// TIA Portal V17 program export: 2 tag tables, 2 data types, 1 data blocks, 3 code blocks (in call order from the OBs), 2 instance data blocks

VAR_GLOBAL   // PLC tag table "Default tag table"
   Clock_Byte AT %MB0 : Byte;
   Clock_10Hz AT %M0.0 : Bool;
   Clock_5Hz AT %M0.1 : Bool;
   "Clock_2.5Hz" AT %M0.2 : Bool;
   Clock_2Hz AT %M0.3 : Bool;
   "Clock_1.25Hz" AT %M0.4 : Bool;
   Clock_1Hz AT %M0.5 : Bool;
   "Clock_0.625Hz" AT %M0.6 : Bool;
   "Clock_0.5Hz" AT %M0.7 : Bool;
END_VAR

VAR_GLOBAL   // PLC tag table "OPC_StatusCodes"
END_VAR
VAR_GLOBAL CONSTANT   // user constants
   OpcUa_Good : DWord := 16#00000000;   // Everything is as expected.
   OpcUa_Uncertain : DWord := 16#40000000;   // Something unexpected occurred but the results still maybe useable.
   OpcUa_Bad : DWord := 16#80000000;   // An error occurred.
   OpcUa_BadUnexpectedError : DWord := 16#80010000;   // An unexpected error occurred.
   OpcUa_BadInternalError : DWord := 16#80020000;   // An internal error occurred as a result of a programming or configuration error.
   OpcUa_BadOutOfMemory : DWord := 16#80030000;   // Not enough memory to complete the operation.
   OpcUa_BadResourceUnavailable : DWord := 16#80040000;   // An operating system resource is not available.
   OpcUa_BadCommunicationError : DWord := 16#80050000;   // A low level communication error occurred.
   OpcUa_BadEncodingError : DWord := 16#80060000;   // Encoding halted because of invalid data in the objects being serialized.
   OpcUa_BadDecodingError : DWord := 16#80070000;   // Decoding halted because of invalid data in the stream.
   OpcUa_BadEncodingLimitsExceeded : DWord := 16#80080000;   // The message encoding/decoding limits imposed by the stack have been exceeded.
   OpcUa_BadRequestTooLarge : DWord := 16#80B80000;   // The request message size exceeds limits set by the server.
   OpcUa_BadResponseTooLarge : DWord := 16#80B90000;   // The response message size exceeds limits set by the client.
   OpcUa_BadUnknownResponse : DWord := 16#80090000;   // An unrecognized response was received from the server.
   OpcUa_BadTimeout : DWord := 16#800A0000;   // The operation timed out.
   OpcUa_BadServiceUnsupported : DWord := 16#800B0000;   // The server does not support the requested service.
   OpcUa_BadShutdown : DWord := 16#800C0000;   // The operation was cancelled because the application is shutting down.
   OpcUa_BadServerNotConnected : DWord := 16#800D0000;   // The operation could not complete because the client is not connected to the server.
   OpcUa_BadServerHalted : DWord := 16#800E0000;   // The server has stopped and cannot process any requests.
   OpcUa_BadNothingToDo : DWord := 16#800F0000;   // There was nothing to do because the client passed a list of operations with no elements.
   OpcUa_BadTooManyOperations : DWord := 16#80100000;   // The request could not be processed because it specified too many operations.
   OpcUa_BadTooManyMonitoredItems : DWord := 16#80DB0000;   // The request could not be processed because there are too many monitored items in the subscription.
   OpcUa_BadDataTypeIdUnknown : DWord := 16#80110000;   // The extension object cannot be (de)serialized because the data type id is not recognized.
   OpcUa_BadCertificateInvalid : DWord := 16#80120000;   // The certificate provided as a parameter is not valid.
   OpcUa_BadSecurityChecksFailed : DWord := 16#80130000;   // An error occurred verifying security.
   OpcUa_BadCertificateTimeInvalid : DWord := 16#80140000;   // The certificate has expired or is not yet valid.
   OpcUa_BadCertificateIssuerTimeInvalid : DWord := 16#80150000;   // An issuer certificate has expired or is not yet valid.
   OpcUa_BadCertificateHostNameInvalid : DWord := 16#80160000;   // The HostName used to connect to a server does not match a HostName in the certificate.
   OpcUa_BadCertificateUriInvalid : DWord := 16#80170000;   // The URI specified in the ApplicationDescription does not match the URI in the certificate.
   OpcUa_BadCertificateUseNotAllowed : DWord := 16#80180000;   // The certificate may not be used for the requested operation.
   OpcUa_BadCertificateIssuerUseNotAllowed : DWord := 16#80190000;   // The issuer certificate may not be used for the requested operation.
   OpcUa_BadCertificateUntrusted : DWord := 16#801A0000;   // The certificate is not trusted.
   OpcUa_BadCertificateRevocationUnknown : DWord := 16#801B0000;   // It was not possible to determine if the certificate has been revoked.
   OpcUa_BadCertificateIssuerRevocationUnknown : DWord := 16#801C0000;   // It was not possible to determine if the issuer certificate has been revoked.
   OpcUa_BadCertificateRevoked : DWord := 16#801D0000;   // The certificate has been revoked.
   OpcUa_BadCertificateIssuerRevoked : DWord := 16#801E0000;   // The issuer certificate has been revoked.
   OpcUa_BadCertificateChainIncomplete : DWord := 16#810D0000;   // The certificate chain is incomplete.
   OpcUa_BadUserAccessDenied : DWord := 16#801F0000;   // User does not have permission to perform the requested operation.
   OpcUa_BadIdentityTokenInvalid : DWord := 16#80200000;   // The user identity token is not valid.
   OpcUa_BadIdentityTokenRejected : DWord := 16#80210000;   // The user identity token is valid but the server has rejected it.
   OpcUa_BadSecureChannelIdInvalid : DWord := 16#80220000;   // The specified secure channel is no longer valid.
   OpcUa_BadInvalidTimestamp : DWord := 16#80230000;   // The timestamp is outside the range allowed by the server.
   OpcUa_BadNonceInvalid : DWord := 16#80240000;   // The nonce does appear to be not a random value or it is not the correct length.
   OpcUa_BadSessionIdInvalid : DWord := 16#80250000;   // The session id is not valid.
   OpcUa_BadSessionClosed : DWord := 16#80260000;   // The session was closed by the client.
   OpcUa_BadSessionNotActivated : DWord := 16#80270000;   // The session cannot be used because ActivateSession has not been called.
   OpcUa_BadSubscriptionIdInvalid : DWord := 16#80280000;   // The subscription id is not valid.
   OpcUa_BadRequestHeaderInvalid : DWord := 16#802A0000;   // The header for the request is missing or invalid.
   OpcUa_BadTimestampsToReturnInvalid : DWord := 16#802B0000;   // The timestamps to return parameter is invalid.
   OpcUa_BadRequestCancelledByClient : DWord := 16#802C0000;   // The request was cancelled by the client.
   OpcUa_BadTooManyArguments : DWord := 16#80E50000;   // Too many arguments were provided.
   OpcUa_BadLicenseExpired : DWord := 16#810E0000;   // The server requires a license to operate in general or to perform a service or operation, but existing license is expired.
   OpcUa_BadLicenseLimitsExceeded : DWord := 16#810F0000;   // The server has limits on number of allowed operations / objects, based on installed licenses, and these limits where exceeded.
   OpcUa_BadLicenseNotAvailable : DWord := 16#81100000;   // The server does not have a license which is required to operate in general or to perform a service or operation.
   OpcUa_GoodSubscriptionTransferred : DWord := 16#002D0000;   // The subscription was transferred to another session.
   OpcUa_GoodCompletesAsynchronously : DWord := 16#002E0000;   // The processing will complete asynchronously.
   OpcUa_GoodOverload : DWord := 16#002F0000;   // Sampling has slowed down due to resource limitations.
   OpcUa_GoodClamped : DWord := 16#00300000;   // The value written was accepted but was clamped.
   OpcUa_BadNoCommunication : DWord := 16#80310000;   // Communication with the data source is defined, but not established, and there is no last known value available.
   OpcUa_BadWaitingForInitialData : DWord := 16#80320000;   // Waiting for the server to obtain values from the underlying data source.
   OpcUa_BadNodeIdInvalid : DWord := 16#80330000;   // The syntax of the node id is not valid.
   OpcUa_BadNodeIdUnknown : DWord := 16#80340000;   // The node id refers to a node that does not exist in the server address space.
   OpcUa_BadAttributeIdInvalid : DWord := 16#80350000;   // The attribute is not supported for the specified Node.
   OpcUa_BadIndexRangeInvalid : DWord := 16#80360000;   // The syntax of the index range parameter is invalid.
   OpcUa_BadIndexRangeNoData : DWord := 16#80370000;   // No data exists within the range of indexes specified.
   OpcUa_BadDataEncodingInvalid : DWord := 16#80380000;   // The data encoding is invalid.
   OpcUa_BadDataEncodingUnsupported : DWord := 16#80390000;   // The server does not support the requested data encoding for the node.
   OpcUa_BadNotReadable : DWord := 16#803A0000;   // The access level does not allow reading or subscribing to the Node.
   OpcUa_BadNotWritable : DWord := 16#803B0000;   // The access level does not allow writing to the Node.
   OpcUa_BadOutOfRange : DWord := 16#803C0000;   // The value was out of range.
   OpcUa_BadNotSupported : DWord := 16#803D0000;   // The requested operation is not supported.
   OpcUa_BadNotFound : DWord := 16#803E0000;   // A requested item was not found or a search operation ended without success.
   OpcUa_BadObjectDeleted : DWord := 16#803F0000;   // The object cannot be used because it has been deleted.
   OpcUa_BadNotImplemented : DWord := 16#80400000;   // Requested operation is not implemented.
   OpcUa_BadMonitoringModeInvalid : DWord := 16#80410000;   // The monitoring mode is invalid.
   OpcUa_BadMonitoredItemIdInvalid : DWord := 16#80420000;   // The monitoring item id does not refer to a valid monitored item.
   OpcUa_BadMonitoredItemFilterInvalid : DWord := 16#80430000;   // The monitored item filter parameter is not valid.
   OpcUa_BadMonitoredItemFilterUnsupported : DWord := 16#80440000;   // The server does not support the requested monitored item filter.
   OpcUa_BadFilterNotAllowed : DWord := 16#80450000;   // A monitoring filter cannot be used in combination with the attribute specified.
   OpcUa_BadStructureMissing : DWord := 16#80460000;   // A mandatory structured parameter was missing or null.
   OpcUa_BadEventFilterInvalid : DWord := 16#80470000;   // The event filter is not valid.
   OpcUa_BadContentFilterInvalid : DWord := 16#80480000;   // The content filter is not valid.
   OpcUa_BadFilterOperatorInvalid : DWord := 16#80C10000;   // An unregognized operator was provided in a filter.
   OpcUa_BadFilterOperatorUnsupported : DWord := 16#80C20000;   // A valid operator was provided, but the server does not provide support for this filter operator.
   OpcUa_BadFilterOperandCountMismatch : DWord := 16#80C30000;   // The number of operands provided for the filter operator was less then expected for the operand provided.
   OpcUa_BadFilterOperandInvalid : DWord := 16#80490000;   // The operand used in a content filter is not valid.
   OpcUa_BadFilterElementInvalid : DWord := 16#80C40000;   // The referenced element is not a valid element in the content filter.
   OpcUa_BadFilterLiteralInvalid : DWord := 16#80C50000;   // The referenced literal is not a valid value.
   OpcUa_BadContinuationPointInvalid : DWord := 16#804A0000;   // The continuation point provide is longer valid.
   OpcUa_BadNoContinuationPoints : DWord := 16#804B0000;   // The operation could not be processed because all continuation points have been allocated.
   OpcUa_BadReferenceTypeIdInvalid : DWord := 16#804C0000;   // The operation could not be processed because all continuation points have been allocated.
   OpcUa_BadBrowseDirectionInvalid : DWord := 16#804D0000;   // The browse direction is not valid.
   OpcUa_BadNodeNotInView : DWord := 16#804E0000;   // The node is not part of the view.
   OpcUa_BadNumericOverflow : DWord := 16#81120000;   // The number was not accepted because of a numeric overflow.
   OpcUa_BadServerUriInvalid : DWord := 16#804F0000;   // The ServerUri is not a valid URI.
   OpcUa_BadServerNameMissing : DWord := 16#80500000;   // No ServerName was specified.
   OpcUa_BadDiscoveryUrlMissing : DWord := 16#80510000;   // No DiscoveryUrl was specified.
   OpcUa_BadSempahoreFileMissing : DWord := 16#80520000;   // The semaphore file specified by the client is not valid.
   OpcUa_BadRequestTypeInvalid : DWord := 16#80530000;   // The security token request type is not valid.
   OpcUa_BadSecurityModeRejected : DWord := 16#80540000;   // The security mode does not meet the requirements set by the server.
   OpcUa_BadSecurityPolicyRejected : DWord := 16#80550000;   // The security policy does not meet the requirements set by the server.
   OpcUa_BadTooManySessions : DWord := 16#80560000;   // The server has reached its maximum number of sessions.
   OpcUa_BadUserSignatureInvalid : DWord := 16#80570000;   // The user token signature is missing or invalid.
   OpcUa_BadApplicationSignatureInvalid : DWord := 16#80580000;   // The signature generated with the client certificate is missing or invalid.
   OpcUa_BadNoValidCertificates : DWord := 16#80590000;   // The client did not provide at least one software certificate that is valid and meets the profile requirements for the server.
   OpcUa_BadIdentityChangeNotSupported : DWord := 16#80C60000;   // The server does not support changing the user identity assigned to the session.
   OpcUa_BadRequestCancelledByRequest : DWord := 16#805A0000;   // The request was cancelled by the client with the Cancel service.
   OpcUa_BadParentNodeIdInvalid : DWord := 16#805B0000;   // The parent node id does not to refer to a valid node.
   OpcUa_BadReferenceNotAllowed : DWord := 16#805C0000;   // The reference could not be created because it violates constraints imposed by the data model.
   OpcUa_BadNodeIdRejected : DWord := 16#805D0000;   // The requested node id was reject because it was either invalid or server does not allow node ids to be specified by the client.
   OpcUa_BadNodeIdExists : DWord := 16#805E0000;   // The requested node id is already used by another node.
   OpcUa_BadNodeClassInvalid : DWord := 16#805F0000;   // The node class is not valid.
   OpcUa_BadBrowseNameInvalid : DWord := 16#80600000;   // The browse name is invalid.
   OpcUa_BadBrowseNameDuplicated : DWord := 16#80610000;   // The browse name is not unique among nodes that share the same relationship with the parent.
   OpcUa_BadNodeAttributesInvalid : DWord := 16#80620000;   // The node attributes are not valid for the node class.
   OpcUa_BadTypeDefinitionInvalid : DWord := 16#80630000;   // The type definition node id does not reference an appropriate type node.
   OpcUa_BadSourceNodeIdInvalid : DWord := 16#80640000;   // The source node id does not reference a valid node.
   OpcUa_BadTargetNodeIdInvalid : DWord := 16#80650000;   // The target node id does not reference a valid node.
   OpcUa_BadDuplicateReferenceNotAllowed : DWord := 16#80660000;   // The reference type between the nodes is already defined.
   OpcUa_BadInvalidSelfReference : DWord := 16#80670000;   // The server does not allow this type of self reference on this node.
   OpcUa_BadReferenceLocalOnly : DWord := 16#80680000;   // The reference type is not valid for a reference to a remote server.
   OpcUa_BadNoDeleteRights : DWord := 16#80690000;   // The server will not allow the node to be deleted.
   OpcUa_UncertainReferenceNotDeleted : DWord := 16#40BC0000;   // The server was not able to delete all target references.
   OpcUa_BadServerIndexInvalid : DWord := 16#806A0000;   // The server index is not valid.
   OpcUa_BadViewIdUnknown : DWord := 16#806B0000;   // The view id does not refer to a valid view node.
   OpcUa_BadViewTimestampInvalid : DWord := 16#80C90000;   // The view timestamp is not available or not supported.
   OpcUa_BadViewParameterMismatch : DWord := 16#80CA0000;   // The view parameters are not consistent with each other.
   OpcUa_BadViewVersionInvalid : DWord := 16#80CB0000;   // The view version is not available or not supported.
   OpcUa_UncertainNotAllNodesAvailable : DWord := 16#40C00000;   // The list of references may not be complete because the underlying system is not available.
   OpcUa_GoodResultsMayBeIncomplete : DWord := 16#00BA0000;   // The server should have followed a reference to a node in a remote server but did not. The result set may be incomplete.
   OpcUa_BadNotTypeDefinition : DWord := 16#80C80000;   // The provided Nodeid was not a type definition nodeid.
   OpcUa_UncertainReferenceOutOfServer : DWord := 16#406C0000;   // One of the references to follow in the relative path references to a node in the address space in another server.
   OpcUa_BadTooManyMatches : DWord := 16#806D0000;   // The requested operation has too many matches to return.
   OpcUa_BadQueryTooComplex : DWord := 16#806E0000;   // The requested operation requires too many resources in the server.
   OpcUa_BadNoMatch : DWord := 16#806F0000;   // The requested operation has no match to return.
   OpcUa_BadMaxAgeInvalid : DWord := 16#80700000;   // The max age parameter is invalid.
   OpcUa_BadSecurityModeInsufficient : DWord := 16#80E60000;   // The operation is not permitted over the current secure channel.
   OpcUa_BadHistoryOperationInvalid : DWord := 16#80710000;   // The history details parameter is not valid.
   OpcUa_BadHistoryOperationUnsupported : DWord := 16#80720000;   // The server does not support the requested operation.
   OpcUa_BadInvalidTimestampArgument : DWord := 16#80BD0000;   // The defined timestamp to return was invalid.
   OpcUa_BadWriteNotSupported : DWord := 16#80730000;   // The server does not support writing the combination of value, status and timestamps provided.
   OpcUa_BadTypeMismatch : DWord := 16#80740000;   // The value supplied for the attribute is not of the same type as the attributes value.
   OpcUa_BadMethodInvalid : DWord := 16#80750000;   // The method id does not refer to a method for the specified object.
   OpcUa_BadArgumentsMissing : DWord := 16#80760000;   // The client did not specify all of the input arguments for the method.
   OpcUa_BadNotExecutable : DWord := 16#81110000;   // The executable attribute does not allow the execution of the method.
   OpcUa_BadTooManySubscriptions : DWord := 16#80770000;   // The server has reached its maximum number of subscriptions.
   OpcUa_BadTooManyPublishRequests : DWord := 16#80780000;   // The server has reached the maximum number of queued publish requests.
   OpcUa_BadNoSubscription : DWord := 16#80790000;   // There is no subscription available for this session.
   OpcUa_BadSequenceNumberUnknown : DWord := 16#807A0000;   // The sequence number is unknown to the server.
   OpcUa_BadMessageNotAvailable : DWord := 16#807B0000;   // The requested notification message is no longer available.
   OpcUa_BadInsufficientClientProfile : DWord := 16#807C0000;   // The client of the current session does not support one or more Profiles that are necessary for the subscription.
   OpcUa_BadStateNotActive : DWord := 16#80BF0000;   // The sub-state machine is not currently active.
   OpcUa_BadTcpServerTooBusy : DWord := 16#807D0000;   // The server cannot process the request because it is too busy.
   OpcUa_BadTcpMessageTypeInvalid : DWord := 16#807E0000;   // The type of the message specified in the header invalid.
   OpcUa_BadTcpSecureChannelUnknown : DWord := 16#807F0000;   // The SecureChannelId and/or TokenId are not currently in use.
   OpcUa_BadTcpMessageTooLarge : DWord := 16#80800000;   // The size of the message specified in the header is too large.
   OpcUa_BadTcpNotEnoughResources : DWord := 16#80810000;   // There are not enough resources to process the request.
   OpcUa_BadTcpInternalError : DWord := 16#80820000;   // An internal error occurred.
   OpcUa_BadTcpEndpointUrlInvalid : DWord := 16#80830000;   // The server does not recognize the QueryString specified.
   OpcUa_BadRequestInterrupted : DWord := 16#80840000;   // The request could not be sent because of a network interruption.
   OpcUa_BadRequestTimeout : DWord := 16#80850000;   // Timeout occurred while processing the request.
   OpcUa_BadSecureChannelClosed : DWord := 16#80860000;   // The secure channel has been closed.
   OpcUa_BadSecureChannelTokenUnknown : DWord := 16#80870000;   // The token has expired or is not recognized.
   OpcUa_BadSequenceNumberInvalid : DWord := 16#80880000;   // The sequence number is not valid.
   OpcUa_BadProtocolVersionUnsupported : DWord := 16#80BE0000;   // The applications do not have compatible protocol versions.
   OpcUa_BadConfigurationError : DWord := 16#80890000;   // There is a problem with the configuration that affects the usefulness of the value.
   OpcUa_BadNotConnected : DWord := 16#808A0000;   // The variable should receive its value from another variable, but has never been configured to do so.
   OpcUa_BadDeviceFailure : DWord := 16#808B0000;   // There has been a failure in the device/data source that generates the value that has affected the value.
   OpcUa_BadSensorFailure : DWord := 16#808C0000;   // There has been a failure in the sensor from which the value is derived by the device/data source.
   OpcUa_BadOutOfService : DWord := 16#808D0000;   // The source of the data is not operational.
   OpcUa_BadDeadbandFilterInvalid : DWord := 16#808E0000;   // The deadband filter is not valid.
   OpcUa_UncertainNoCommunicationLastUsableValue : DWord := 16#408F0000;   // Communication to the data source has failed. The variable value is the last value that had a good quality.
   OpcUa_UncertainLastUsableValue : DWord := 16#40900000;   // Whatever was updating this value has stopped doing so.
   OpcUa_UncertainSubstituteValue : DWord := 16#40910000;   // The value is an operational value that was manually overwritten.
   OpcUa_UncertainInitialValue : DWord := 16#40920000;   // The value is an initial value for a variable that normally receives its value from another variable.
   OpcUa_UncertainSensorNotAccurate : DWord := 16#40930000;   // The value is at one of the sensor limits.
   OpcUa_UncertainEngineeringUnitsExceeded : DWord := 16#40940000;   // The value is outside of the range of values defined for this parameter.
   OpcUa_UncertainSubNormal : DWord := 16#40950000;   // The value is derived from multiple sources and has less than the required number of Good sources.
   OpcUa_GoodLocalOverride : DWord := 16#00960000;   // The value has been overridden.
   OpcUa_BadRefreshInProgress : DWord := 16#80970000;   // This Condition refresh failed, a Condition refresh operation is already in progress.
   OpcUa_BadConditionAlreadyDisabled : DWord := 16#80980000;   // This condition has already been disabled.
   OpcUa_BadConditionAlreadyEnabled : DWord := 16#80CC0000;   // This condition has already been enabled.
   OpcUa_BadConditionDisabled : DWord := 16#80990000;   // Property not available, this condition is disabled.
   OpcUa_BadEventIdUnknown : DWord := 16#809A0000;   // The specified event id is not recognized.
   OpcUa_BadEventNotAcknowledgeable : DWord := 16#80BB0000;   // The event cannot be acknowledged.
   OpcUa_BadDialogNotActive : DWord := 16#80CD0000;   // The dialog condition is not active.
   OpcUa_BadDialogResponseInvalid : DWord := 16#80CE0000;   // The response is not valid for the dialog.
   OpcUa_BadConditionBranchAlreadyAcked : DWord := 16#80CF0000;   // The condition branch has already been acknowledged.
   OpcUa_BadConditionBranchAlreadyConfirmed : DWord := 16#80D00000;   // The condition branch has already been confirmed.
   OpcUa_BadConditionAlreadyShelved : DWord := 16#80D10000;   // The condition has already been shelved.
   OpcUa_BadConditionNotShelved : DWord := 16#80D20000;   // The condition is not currently shelved.
   OpcUa_BadShelvingTimeOutOfRange : DWord := 16#80D30000;   // The shelving time not within an acceptable range.
   OpcUa_BadNoData : DWord := 16#809B0000;   // No data exists for the requested time range or event filter.
   OpcUa_BadBoundNotFound : DWord := 16#80D70000;   // No data found to provide upper or lower bound value.
   OpcUa_BadBoundNotSupported : DWord := 16#80D80000;   // The server cannot retrieve a bound for the variable.
   OpcUa_BadDataLost : DWord := 16#809D0000;   // Data is missing due to collection started/stopped/lost.
   OpcUa_BadDataUnavailable : DWord := 16#809E0000;   // Expected data is unavailable for the requested time range due to an un-mounted volume, an off-line archive or tape, or similar reason for temporary unavailability.
   OpcUa_BadEntryExists : DWord := 16#809F0000;   // The data or event was not successfully inserted because a matching entry exists.
   OpcUa_BadNoEntryExists : DWord := 16#80A00000;   // The data or event was not successfully updated because no matching entry exists.
   OpcUa_BadTimestampNotSupported : DWord := 16#80A10000;   // The client requested history using a timestamp format the server does not support (i.e requested ServerTimestamp when server only supports SourceTimestamp).
   OpcUa_GoodEntryInserted : DWord := 16#00A20000;   // The data or event was successfully inserted into the historical database.
   OpcUa_GoodEntryReplaced : DWord := 16#00A30000;   // The data or event field was successfully replaced in the historical database.
   OpcUa_UncertainDataSubNormal : DWord := 16#40A40000;   // The value is derived from multiple values and has less than the required number of Good values.
   OpcUa_GoodNoData : DWord := 16#00A50000;   // No data exists for the requested time range or event filter.
   OpcUa_GoodMoreData : DWord := 16#00A60000;   // The data or event field was successfully replaced in the historical database.
   OpcUa_BadAggregateListMismatch : DWord := 16#80D40000;   // The requested number of Aggregates does not match the requested number of NodeIds.
   OpcUa_BadAggregateNotSupported : DWord := 16#80D50000;   // The requested Aggregate is not support by the server.
   OpcUa_BadAggregateInvalidInputs : DWord := 16#80D60000;   // The aggregate value could not be derived due to invalid data inputs.
   OpcUa_BadAggregateConfigurationRejected : DWord := 16#80DA0000;   // The aggregate configuration is not valid for specified node.
   OpcUa_GoodDataIgnored : DWord := 16#00D90000;   // The request pecifies fields which are not valid for the EventType or cannot be saved by the historian.
   OpcUa_BadRequestNotAllowed : DWord := 16#80E40000;   // The request was rejected by the server because it did not meet the criteria set by the server.
   OpcUa_BadRequestNotComplete : DWord := 16#81130000;   // The request has not been processed by the server yet.
   OpcUa_GoodEdited : DWord := 16#00DC0000;   // The value does not come from the real source and has been edited by the server.
   OpcUa_GoodPostActionFailed : DWord := 16#00DD0000;   // There was an error in execution of these post-actions.
   OpcUa_UncertainDominantValueChanged : DWord := 16#40DE0000;   // The related EngineeringUnit has been changed but the Variable Value is still provided based on the previous unit.
   OpcUa_GoodDependentValueChanged : DWord := 16#00E00000;   // A dependent value has been changed but the change has not been applied to the device.
   OpcUa_BadDominantValueChanged : DWord := 16#80E10000;   // The related EngineeringUnit has been changed but this change has not been applied to the device. The Variable Value is still dependent on the previous unit but its status is currently Bad.
   OpcUa_UncertainDependentValueChanged : DWord := 16#40E20000;   // A dependent value has been changed but the change has not been applied to the device. The quality of the dominant variable is uncertain.
   OpcUa_BadDependentValueChanged : DWord := 16#80E30000;   // A dependent value has been changed but the change has not been applied to the device. The quality of the dominant variable is Bad.
   OpcUa_GoodCommunicationEvent : DWord := 16#00A70000;   // The communication layer has raised an event.
   OpcUa_GoodShutdownEvent : DWord := 16#00A80000;   // The system is shutting down.
   OpcUa_GoodCallAgain : DWord := 16#00A90000;   // The operation is not finished and needs to be called again.
   OpcUa_GoodNonCriticalTimeout : DWord := 16#00AA0000;   // A non-critical timeout occurred.
   OpcUa_BadInvalidArgument : DWord := 16#80AB0000;   // One or more arguments are invalid.
   OpcUa_BadConnectionRejected : DWord := 16#80AC0000;   // Could not establish a network connection to remote server.
   OpcUa_BadDisconnect : DWord := 16#80AD0000;   // The server has disconnected from the client.
   OpcUa_BadConnectionClosed : DWord := 16#80AE0000;   // The network connection has been closed.
   OpcUa_BadInvalidState : DWord := 16#80AF0000;   // The operation cannot be completed because the object is closed, uninitialized or in some other invalid state.
   OpcUa_BadEndOfStream : DWord := 16#80B00000;   // Cannot move beyond end of the stream.
   OpcUa_BadNoDataAvailable : DWord := 16#80B10000;   // No data is currently available for reading from a non-blocking stream.
   OpcUa_BadWaitingForResponse : DWord := 16#80B20000;   // The asynchronous operation is waiting for a response.
   OpcUa_BadOperationAbandoned : DWord := 16#80B30000;   // The asynchronous operation was abandoned by the caller.
   OpcUa_BadExpectedStreamToBlock : DWord := 16#80B40000;   // The stream did not return all data requested (possibly because it is a non-blocking stream).
   OpcUa_BadWouldBlock : DWord := 16#80B50000;   // Non blocking behaviour is required and the operation would block.
   OpcUa_BadSyntaxError : DWord := 16#80B60000;   // A value had an invalid syntax.
   OpcUa_BadMaxConnectionsReached : DWord := 16#80B70000;   // The operation could not be finished because all available connections are in use.
END_VAR

TYPE "typeOPCUAMethodHandling"
// stored: IsFailsafeCompliant false
   STRUCT
      Called : Bool;
      Finished : Bool;
      Result : DWord;
   END_STRUCT;
END_TYPE

TYPE "typeOPCUAStatus"
// stored: IsFailsafeCompliant false
   STRUCT
      done : Bool;
      busy : Bool;
      error : Bool;
      status : DWord;
   END_STRUCT;
END_TYPE

DATA_BLOCK "OpcUaInterface"   // DB31
{ S7_Optimized_Access := 'TRUE' }
VERSION : 0.1
// stored: AutoNumber false, DBAccessibleFromOPCUA true, DBAccessibleFromWebserver true, IsOnlyStoredInLoadMemory false, IsRetainMemResEnabled false, IsWriteProtectedInAS false, MemoryReserve 100
   VAR
      startCounting : Bool;
      endValue : DInt := 10;
      actValue { ExternalWritable := 'False'} : DInt;
      valueResetted { ExternalAccessible := 'False'; ExternalVisible := 'False'; ExternalWritable := 'False'} : Bool;
   END_VAR
BEGIN
END_DATA_BLOCK

ORGANIZATION_BLOCK "Main"   // OB1, LAD, ProgramCycle
TITLE = "Main Program Sweep (Cycle)"
{ S7_Optimized_Access := 'TRUE' }
VERSION : 0.1
// stored: AutoNumber true, IsIECCheckEnabled false, SetENOAutomatically false
   VAR_INPUT
      Initial_Call : Bool;   // Initial call of this OB
      Remanence : Bool;   // =True, if remanent data are available
   END_VAR
BEGIN

REGION Network 1
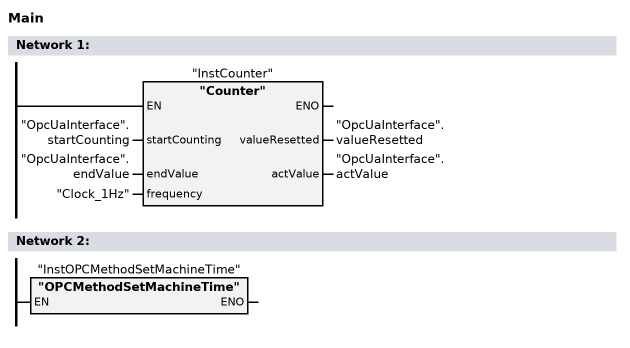
   RUNG wire#powerrail
      "InstCounter"(startCounting := "OpcUaInterface".startCounting, endValue := "OpcUaInterface".endValue, frequency := "Clock_1Hz", valueResetted => "OpcUaInterface".valueResetted, actValue => "OpcUaInterface".actValue)
   END_RUNG
   // the same network as SCL:
   "InstCounter"(startCounting := "OpcUaInterface".startCounting,   // "Counter"
                 endValue := "OpcUaInterface".endValue,
                 frequency := "Clock_1Hz",
                 valueResetted => "OpcUaInterface".valueResetted,
                 actValue => "OpcUaInterface".actValue);
END_REGION

REGION Network 2
   RUNG wire#powerrail
      "InstOPCMethodSetMachineTime"()
   END_RUNG
   // the same network as SCL:
   "InstOPCMethodSetMachineTime"();   // "OPCMethodSetMachineTime"
END_REGION
END_ORGANIZATION_BLOCK

FUNCTION_BLOCK "Counter"
{ S7_Optimized_Access := 'TRUE' }
VERSION : 0.1
   VAR_INPUT 
      startCounting { ExternalWritable := 'False'} : Bool;
      endValue : DInt := 10;
      frequency : Bool;
   END_VAR

   VAR_OUTPUT 
      valueResetted { ExternalWritable := 'False'} : Bool;
      actValue { ExternalWritable := 'False'} : DInt;
   END_VAR

   VAR 
      statValue : DInt;
      statEndValue : DInt;
      InstRTrig {InstructionName := 'R_TRIG'; LibVersion := '1.0'} : R_TRIG;
      statFreqTrig : Bool;
   END_VAR


BEGIN
	IF #startCounting THEN
	    //start counting after user program triggers
	    #InstRTrig(CLK:=#frequency,
	               Q=>#statFreqTrig);
	    #statEndValue := #endValue;
	    IF #statValue <= #statEndValue THEN
	        IF #statFreqTrig THEN
	            #statValue := #statValue + 1;
	            #valueResetted := FALSE;
	        END_IF;
	    ELSE
	        #statValue := 0;
	        #valueResetted := TRUE;
	    END_IF;
	ELSE //no counting
	    //IDLE
	    ;
	END_IF;
	
	#actValue := #statValue;
END_FUNCTION_BLOCK

FUNCTION_BLOCK "OPCMethodSetMachineTime"
{ S7_Optimized_Access := 'TRUE' }
VERSION : 0.1
   VAR 
      OPC_UA_ServerMethodPre_Instance {InstructionName := 'OPC_UA_ServerMethodPre'; LibVersion := '1.0'} : OPC_UA_ServerMethodPre;
      statUAMStatusPre : "typeOPCUAStatus";
      statUAMStatusPost : "typeOPCUAStatus";
      UAMethod_InParameters : Struct
         DateTime : LDT;
      END_STRUCT;
      OPC_UA_ServerMethodPost_Instance {InstructionName := 'OPC_UA_ServerMethodPost'; LibVersion := '1.0'} : OPC_UA_ServerMethodPost;
   END_VAR

   VAR_TEMP 
      tempUAMMethodHandling : "typeOPCUAMethodHandling";
      tempIntReturnOfSysTime : Int;
   END_VAR

   VAR CONSTANT 
      NO_ERROR : Int := 16#0000;
      ERROR_IN_DATE : Int := 16#8080;
      ERROR_IN_TIME : Int := 16#8081;
      REAL_TIME_CLOCK_FAILED : Int := 16#80B0;
   END_VAR


BEGIN
	//=============================================================================
	// Siemens// (c)Copyright (2017)
	//-----------------------------------------------------------------------------
	// Library: -
	// Tested with: CPU:-  FW:-
	// Engineering: TIA Portal (inc 25)
	// Restrictions: -
	// Requirements: OPCUA Server activated, Fimware V2.5
	// Functionality: sets the machine time to a userdefined value.
	//-----------------------------------------------------------------------------
	// Change log table:
	// Version Date Expert in charge Changes applied
	// 04.12.2017 dd.mm.yyyy (APC ERLF) First released version //=============================================================================
	REGION INIT Temp
	    #tempIntReturnOfSysTime := 0;
	    #tempUAMMethodHandling.Called := FALSE;
	    #tempUAMMethodHandling.Finished := FALSE;
	    #tempUAMMethodHandling.Result := "OpcUa_Good";
	END_REGION
	
	REGION PRE
	    #OPC_UA_ServerMethodPre_Instance(Done => #statUAMStatusPre.done,
	                                     Busy => #statUAMStatusPre.busy,
	                                     Error => #statUAMStatusPre.error,
	                                     Status => #statUAMStatusPre.status,
	                                     UAMethod_Called => #tempUAMMethodHandling.Called,
	                                     UAMethod_InParameters := #UAMethod_InParameters);
	END_REGION
	
	REGION FUNCTIONALITY
	    IF #tempUAMMethodHandling.Called THEN
	        #tempIntReturnOfSysTime := WR_SYS_T(#UAMethod_InParameters.DateTime);
	        
	        //ERROR Generation and handling
	        IF #tempIntReturnOfSysTime = #NO_ERROR THEN
	             #tempUAMMethodHandling.Result := "OpcUa_Good";
	        ELSIF #tempIntReturnOfSysTime = #ERROR_IN_DATE THEN
	            #tempUAMMethodHandling.Result := "OpcUa_BadSyntaxError";
	        ELSIF #tempIntReturnOfSysTime = #ERROR_IN_TIME THEN
	            #tempUAMMethodHandling.Result := "OpcUa_BadSyntaxError";
	        ELSIF #tempIntReturnOfSysTime = #REAL_TIME_CLOCK_FAILED THEN
	            #tempUAMMethodHandling.Result := "OpcUa_BadInternalError";
	        END_IF;
	        //SET METHOD TO DONE
	        #tempUAMMethodHandling.Finished := TRUE;
	    END_IF;
	END_REGION
	
	
	REGION Post
	    #OPC_UA_ServerMethodPost_Instance(UAMethod_Result := #tempUAMMethodHandling.Result,
	                                      UAMethod_Finished := #tempUAMMethodHandling.Finished,
	                                      Done => #statUAMStatusPost.done,
	                                      Busy => #statUAMStatusPost.busy,
	                                      Error => #statUAMStatusPost.error,
	                                      Status => #statUAMStatusPost.status);
	END_REGION
END_FUNCTION_BLOCK

DATA_BLOCK "InstCounter"   // DB2
VERSION : 0.1
// stored: AutoNumber true, DBAccessibleFromOPCUA true, DBAccessibleFromWebserver true, InstanceOfName Counter, InstanceOfType FB
"Counter"
BEGIN
END_DATA_BLOCK

DATA_BLOCK "InstOPCMethodSetMachineTime"   // DB3
VERSION : 0.1
// stored: AutoNumber true, DBAccessibleFromOPCUA true, DBAccessibleFromWebserver true, InstanceOfName OPCMethodSetMachineTime, InstanceOfType FB
"OPCMethodSetMachineTime"
BEGIN
END_DATA_BLOCK
